FUNCTION_BLOCK FB_Coordinador_ST
VAR_INPUT
	Tray_1 : BOOL; 
	Tray_2 : BOOL;
END_VAR
VAR_OUTPUT

END_VAR
VAR
	Director : FB_Director_ST;
	Coordinador : FB_Coordinador_SFC;
	Discharger : FB_Discharger_ST;
	ModeAns : GEMMA;
	
END_VAR

Director(IC:= Coordinador.IC, Manual:= Panel.Manual, Go:= Panel.Go, Stop := Panel.Stop,
		 Play := Panel.Play, Cancel := Panel.Stop, EndBatch := Coordinador.Done,
		 End := Panel.End, Fail := Fail);

Panel(Mode := Director.Mode);
		 
Coordinador(IC:=Discharger.IC,
		    Discharger_Execute:=Director.Discharge,
			Discharger_Ready:= Discharger.Ready,
			Discharger_Done:= Discharger.Done,
			Tray_1 := Tray_1,
			Tray_2:= Tray_2);
			
// Associate module variables
Discharger (Execute :=Coordinador.Discharger_Execute,
			Ack := Coordinador.Discharger_Ack,
			Reset := Director.Reset,
			Pause := Director.Pause,
			B1 := Tray_1,
			B2 := Tray_2);

END_FUNCTION_BLOCK

(* stored: Version 1.1.0.1, ProductVersion 3.1.4024.6
   POU FB_Coordinador_ST: Id {30bafdc6-6690-419c-8cbe-ff0c64e369c1}, SpecialFunc None *)
